// TIA Portal V16 export
// export: Created 2025-05-30T16:30:19.2472967Z, ExportSetting WithDefaults, DisplayName Totally Integrated Automation Portal, DisplayVersion V16, DisplayName TIA Portal Version Control Interface, DisplayVersion V16, DisplayName TIA Portal Openness, DisplayVersion V16, DisplayName STEP 7 Professional, DisplayVersion V16, DisplayName STEP 7 Safety, DisplayVersion V16, DisplayName WinCC Advanced, DisplayVersion V16
FUNCTION_BLOCK "ESB_Flash_Warning_Block"   // FB1, FBD
VERSION : 0.1
// stored: AutoNumber true, IsIECCheckEnabled false, UDAEnableTagReadback false
   VAR_INPUT
      "Safety Feedback Contact" : Bool;
      "WarningTimer Time 1" : Time := T#150ms;
      "WarningTimer Time 2" : Time := T#150ms;
   END_VAR
   VAR_OUTPUT
      "Warning Ouput Contact" : Bool;
      "ET WarningTimer 1" : Time;
      "ET WarningTimer 2" : Time;
   END_VAR
   VAR_TEMP
      SafetyTakeoverContact : Bool;
   END_VAR
   VAR_TEMP   // added for the SCL form of the ladder/FBD networks
      _w1 : Bool;
   END_VAR
BEGIN

REGION Network 1: Flash Warning
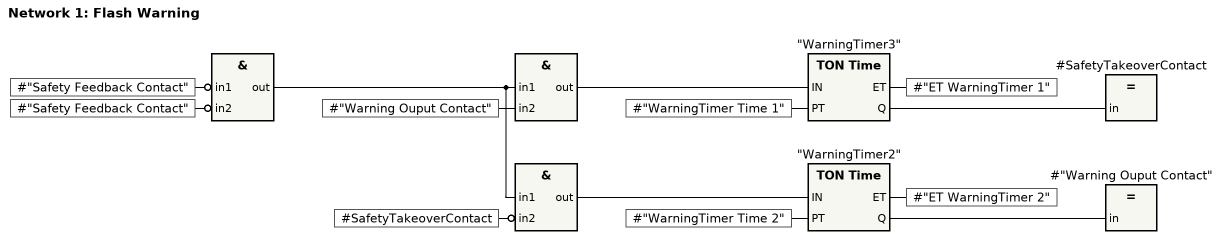
   #_w1 := NOT #"Safety Feedback Contact" AND NOT #"Safety Feedback Contact";
   "WarningTimer3".TON(IN := #_w1 AND #"Warning Ouput Contact",
                       PT := #"WarningTimer Time 1",
                       ET => #"ET WarningTimer 1");
   #SafetyTakeoverContact := "WarningTimer3".Q;
   "WarningTimer2".TON(IN := #_w1 AND NOT #SafetyTakeoverContact,
                       PT := #"WarningTimer Time 2",
                       ET => #"ET WarningTimer 2");
   #"Warning Ouput Contact" := "WarningTimer2".Q;
END_REGION
END_FUNCTION_BLOCK
